Staubli VAL3: testMove.pgx

program testMove()
begin
  bfnshint=true
  //        if bfnshint==true
  //delay(0.0968)
  taskCreateSync "SychMove",0.004,bRes,task_sychron()
  //call task_sychron()
end
